FUNCTION_BLOCK EV3_CONTROLLER (* Service Interface Function Block Type *)
  (* Standard: 61499-2 *)
  (* Version 0.0, 2008-07-10, 4DIAC-IDE, 4DIAC-Consortium *)
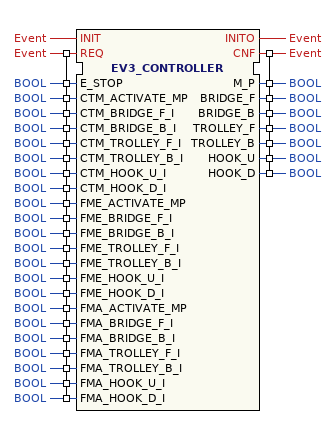
  EVENT_INPUT
    INIT; (* Service Initialization *)
    REQ WITH E_STOP, CTM_ACTIVATE_MP, CTM_BRIDGE_F_I, CTM_BRIDGE_B_I, CTM_TROLLEY_F_I, CTM_TROLLEY_B_I, CTM_HOOK_D_I, CTM_HOOK_U_I, FME_ACTIVATE_MP, FME_BRIDGE_F_I, FME_BRIDGE_B_I, FME_TROLLEY_F_I, FME_TROLLEY_B_I, FME_HOOK_U_I, FME_HOOK_D_I, FMA_ACTIVATE_MP, FMA_BRIDGE_F_I, FMA_BRIDGE_B_I, FMA_TROLLEY_F_I, FMA_TROLLEY_B_I, FMA_HOOK_U_I, FMA_HOOK_D_I; (* Service Request *)
  END_EVENT
  EVENT_OUTPUT
    INITO; (* Initialization Confirm *)
    CNF WITH BRIDGE_F, TROLLEY_F, HOOK_U, M_P, BRIDGE_B, TROLLEY_B, HOOK_D; (* Confirmation of Requested Service *)
  END_EVENT
  VAR_INPUT
    E_STOP : BOOL; (* Emergency controller *)
    CTM_ACTIVATE_MP : BOOL;
    CTM_BRIDGE_F_I : BOOL;
    CTM_BRIDGE_B_I : BOOL;
    CTM_TROLLEY_F_I : BOOL;
    CTM_TROLLEY_B_I : BOOL;
    CTM_HOOK_U_I : BOOL;
    CTM_HOOK_D_I : BOOL;
    FME_ACTIVATE_MP : BOOL;
    FME_BRIDGE_F_I : BOOL;
    FME_BRIDGE_B_I : BOOL;
    FME_TROLLEY_F_I : BOOL;
    FME_TROLLEY_B_I : BOOL;
    FME_HOOK_U_I : BOOL;
    FME_HOOK_D_I : BOOL;
    FMA_ACTIVATE_MP : BOOL;
    FMA_BRIDGE_F_I : BOOL;
    FMA_BRIDGE_B_I : BOOL;
    FMA_TROLLEY_F_I : BOOL;
    FMA_TROLLEY_B_I : BOOL;
    FMA_HOOK_U_I : BOOL;
    FMA_HOOK_D_I : BOOL;
  END_VAR
  VAR_OUTPUT
    M_P : BOOL; (* Motor positions *)
    BRIDGE_F : BOOL;
    BRIDGE_B : BOOL;
    TROLLEY_F : BOOL;
    TROLLEY_B : BOOL;
    HOOK_U : BOOL;
    HOOK_D : BOOL;
  END_VAR
  SERVICE APPLICATION/RESOURCE (* Service Interface Function Block Type *)
    SEQUENCE normal_establishment
      APPLICATION.INIT+(PARAMS) -> RESOURCE.initialize(PARAMS) -> APPLICATION.INITO+();
    END_SEQUENCE
    SEQUENCE unsuccessful_establishment
      APPLICATION.INIT+(PARAMS) -> RESOURCE.initialize(PARAMS) -> APPLICATION.INITO-(STATUS);
    END_SEQUENCE
    SEQUENCE request_confirm
      APPLICATION.REQ+(SD) -> RESOURCE.request(SD) -> APPLICATION.CNF+(RD);
    END_SEQUENCE
    SEQUENCE request_inhibited
      APPLICATION.REQ-(SD) -> APPLICATION.CNF-(STATUS);
    END_SEQUENCE
    SEQUENCE request_error
      APPLICATION.REQ+(SD) -> RESOURCE.request(SD) -> APPLICATION.CNF-(STATUS);
    END_SEQUENCE
    SEQUENCE indication_response
      RESOURCE.indicate(RD) -> APPLICATION.IND+(RD);
      APPLICATION.RSP(QI,SD) -> RESOURCE.response(QI,SD);
    END_SEQUENCE
    SEQUENCE indication_inhibited
      RESOURCE.indicate(RD,QI=FALSE) -> RESOURCE.inhibited();
    END_SEQUENCE
    SEQUENCE error_indication
      RESOURCE.error(STATUS) -> APPLICATION.IND-(STATUS);
    END_SEQUENCE
    SEQUENCE application_initiated_termination
      APPLICATION.INIT-() -> RESOURCE.terminate() -> APPLICATION.INITO-(STATUS);
    END_SEQUENCE
    SEQUENCE resource_initiated_termination
      -> APPLICATION.INITO-(STATUS);
    END_SEQUENCE
  END_SERVICE
END_FUNCTION_BLOCK
